// TIA Portal V19 export
TYPE "A0301_Mach_Ax_Pos_Data"
   STRUCT
      OffsetPosAttesa { S7_SetPoint := 'True'} : LReal;
      PosAttesa { S7_SetPoint := 'True'} : LReal;
      PosFineSpinta { S7_SetPoint := 'True'} : LReal;
   END_STRUCT;
END_TYPE
